PROGRAM MAIN
VAR
	MrAnglef: REAL;
	MrHypotenusef: REAL;
	MrResultat: REAL;
END_VAR

MrResultat:=f_calcul(MrAnglef,MrHypotenusef);

END_PROGRAM

(* stored: Version 1.1.0.1, ProductVersion 3.1.4020.6
   POU MAIN: Id {bc23ed29-a0d3-44c0-9898-2f5e03cb9c88}, SpecialFunc None *)
